KUKA KRL data list: ros_krlptp.dat

&ACCESS RVP
&REL 74
&PARAM DISKPATH = KRC:\R1\Program\ROS
DEFDAT  ROS_KRLPTP PUBLIC
INT movesQueued=0
REAL moveTime=0.200000
REAL moveTime2=0.104000
E6AXIS nextMove={A1 -156.919830,A2 -103.435272,A3 29.4374046,A4 2.74812388,A5 -45.1240845,A6 10.6140194,E1 0.0,E2 0.0,E3 0.0,E4 0.0,E5 0.0,E6 0.0}
DECL PDAT ROS_Pdat={VEL 50.0000,ACC 50.0000,APO_DIST 20.0000,GEAR_JERK 100.000,EXAX_IGN 0}
ENDDAT
